(* Logix 5000 project; controller Transcat_L33ER vendor 1 type 14 code 107 rev 32.11; software revision 32.02; part 4 of 5 *)
(* tags used below, declared in another part *)
   AnyAutoDeviceInterlock : BOOL;   // Any device in Auto interlocked
   AnyAutoRun : BOOL;   // Bit that in on if ANY device is placed into Auto run (to signal pre-start beed)
   AnyDeviceInterlock : BOOL;   // Any device is interlocked
   AnyManualRun : BOOL;   // Bit that in on if ANY device is placed into manual run (to signal pre-start beed)
   Auto_Run_All_Interlock : BOOL;   // Bit to interlock all devices running in Auto
   BeaconBlueLight : ALIAS FOR TC_Remote_IO:3:O.3;   // Blue Beacon Light
   BeaconGreenLight : ALIAS FOR TC_Remote_IO:3:O.2;   // Green Beacon Light
   BeaconRedLight : ALIAS FOR TC_Remote_IO:3:O.0;   // Red Beacon Light
   BeaconYellowLight : ALIAS FOR TC_Remote_IO:3:O.1;   // Yellow Beacon Light
   Beep : BOOL;   // Bit to Activte Beacon Alarm
   BeepNew : ALIAS FOR TC_Remote_IO:3:O.4;
   Device : Device[20];
   EstopActive : BOOL;   // E
   EStopReset_OS : BOOL;   // Storage bit required by the ONS instruction
   EStopResetArmed : BOOL;   // Remembers that Banner entered the waiting-for-reset state
   EStopResetPulse : BOOL;   // One-scan pulse used to clear all 14 E-stop interlocks - allows reset of estop interlocks from physical reset button on V
   FT103 : BronkhorstFlowMeter;
   FT103B : BronkhorstFlowMeter;
   FT104 : BronkhorstFlowMeter;
   FT104B : BronkhorstFlowMeter;
   FT105 : BronkhorstFlowMeter;
   FT105B : BronkhorstFlowMeter;
   GF101 : Thayer_WB_Feeder;   // Thayer 1 Tags
   GF101_Write_Acknowledge : ALIAS FOR Thayer1_BS:O.Data[2].5;   // Thayer 1 (GF101) Acknowledge
   GF201 : Thayer_WB_Feeder;   // Thayer 2 Tags
   GF201_Write_Acknowledge : ALIAS FOR Thayer2_BS:O.Data[2].5;   // Thayer 2 (GF201) Acknowledge
   GreenFlashingOff : TIMER;
   GreenFlashingOn : TIMER;
   HMI_AllReset : BOOL;   // Bit to reset Auto/Man, AutoRun, RecipeRun, TimedRunEnable to 0 from HMI
   HMI_ProcessReset : BOOL;   // Bit to clear the process hold/inteerlock when all other device interlocks are cleared
   MX101 : Howes_Mixer;
   MX201 : Howes_Mixer;
   PT103_PV_RAW : ALIAS FOR TC_Remote_IO:1:I.Ch0Data;   // Raw (unscaled) pressure reading from PT103 - PSI * 100 (range 0 - 108 PSI)
   PT104_PV_RAW : ALIAS FOR TC_Remote_IO:1:I.Ch1Data;   // Raw (unscaled) pressure reading from PT104 - PSI * 100 (range 0 - 108 PSI)
   PT105_PV_RAW : ALIAS FOR TC_Remote_IO:1:I.Ch2Data;   // Raw (unscaled) pressure reading from PT105 - PSI * 100 (range 0 - 108 PSI)
   StartBeepTimer : TIMER;   // Timer to sound the beep alarm before starting a device
   VF101 : Acrison_Feeder;   // Medium Feeder Tags
   VF201 : Acrison_Feeder;   // Small Feeder 2 Tags
   VFD_Panel_Safety_Panel_Etop_OK : ALIAS FOR XS26_VFD_Cabinet_Safety_Controller:I1.Data[1].6;
   VFD_Panel_Safety_Remote_Estops_OK : ALIAS FOR XS26_VFD_Cabinet_Safety_Controller:I1.Data[1].7;
   VFD_Panel_Safety_WaitingForReset : ALIAS FOR XS26_VFD_Cabinet_Safety_Controller:I1.Data[1].5;
   YellowFlashOff : TIMER;
   YellowFlashOn : TIMER;
(* MainProgram, continued *)

ROUTINE InterlockLogic   (* ladder *)
// All interlock logic is handled here
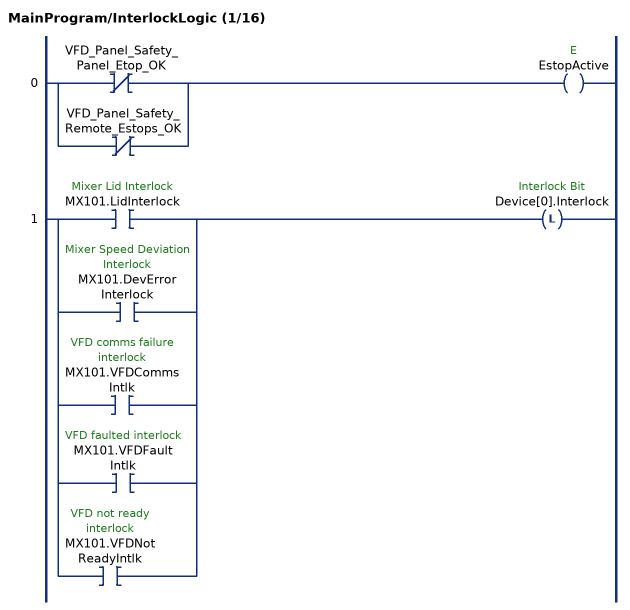
   0: [XIO(VFD_Panel_Safety_Panel_Etop_OK) ,XIO(VFD_Panel_Safety_Remote_Estops_OK) ]OTE(EstopActive);
   1: [XIC(MX101.LidInterlock) ,XIC(MX101.DevErrorInterlock) ,XIC(MX101.VFDCommsIntlk) ,XIC(MX101.VFDFaultIntlk) ,XIC(MX101.VFDNotReadyIntlk) ]OTL(Device[0].Interlock);
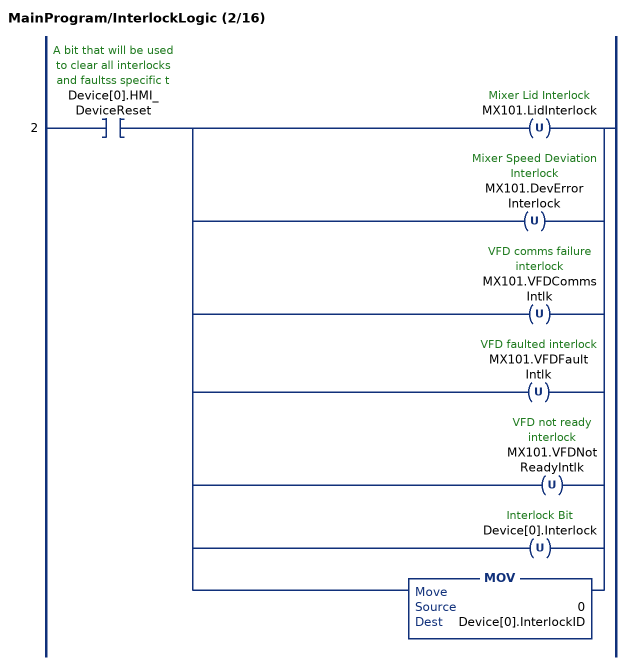
   2: XIC(Device[0].HMI_DeviceReset)[OTU(MX101.LidInterlock) ,OTU(MX101.DevErrorInterlock) ,OTU(MX101.VFDCommsIntlk) ,OTU(MX101.VFDFaultIntlk) ,OTU(MX101.VFDNotReadyIntlk) ,OTU(Device[0].Interlock) ,MOV(0,Device[0].InterlockID) ];
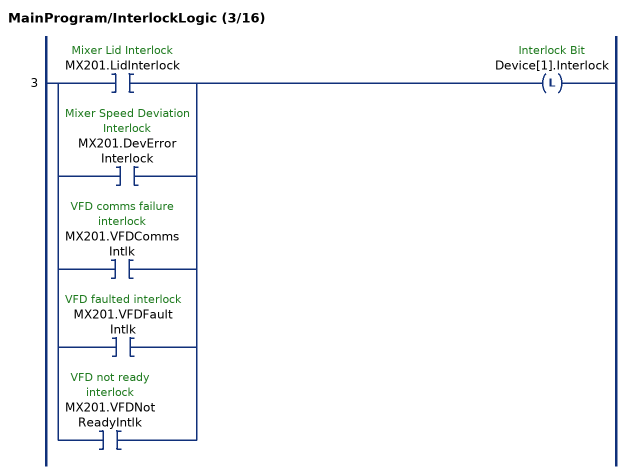
   3: [XIC(MX201.LidInterlock) ,XIC(MX201.DevErrorInterlock) ,XIC(MX201.VFDCommsIntlk) ,XIC(MX201.VFDFaultIntlk) ,XIC(MX201.VFDNotReadyIntlk) ]OTL(Device[1].Interlock);
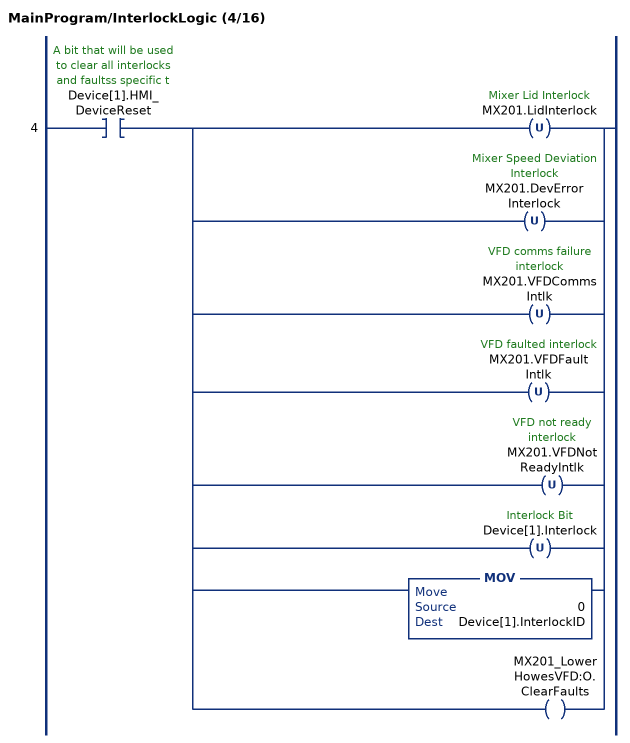
   4: XIC(Device[1].HMI_DeviceReset)[OTU(MX201.LidInterlock) ,OTU(MX201.DevErrorInterlock) ,OTU(MX201.VFDCommsIntlk) ,OTU(MX201.VFDFaultIntlk) ,OTU(MX201.VFDNotReadyIntlk) ,OTU(Device[1].Interlock) ,MOV(0,Device[1].InterlockID) ,OTE(MX201_LowerHowesVFD:O.ClearFaults) ];
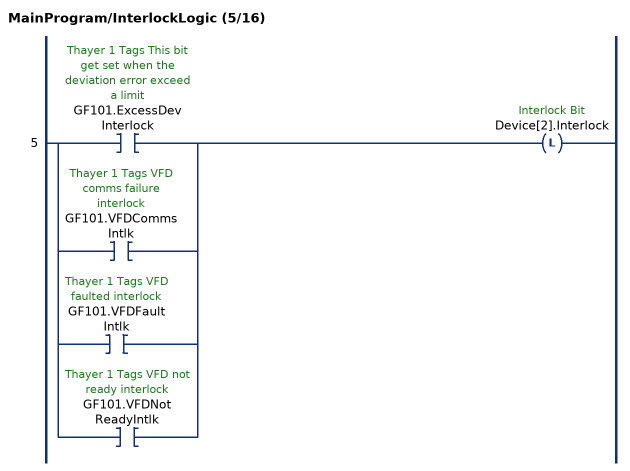
   5: [XIC(GF101.ExcessDevInterlock) ,XIC(GF101.VFDCommsIntlk) ,XIC(GF101.VFDFaultIntlk) ,XIC(GF101.VFDNotReadyIntlk) ]OTL(Device[2].Interlock);
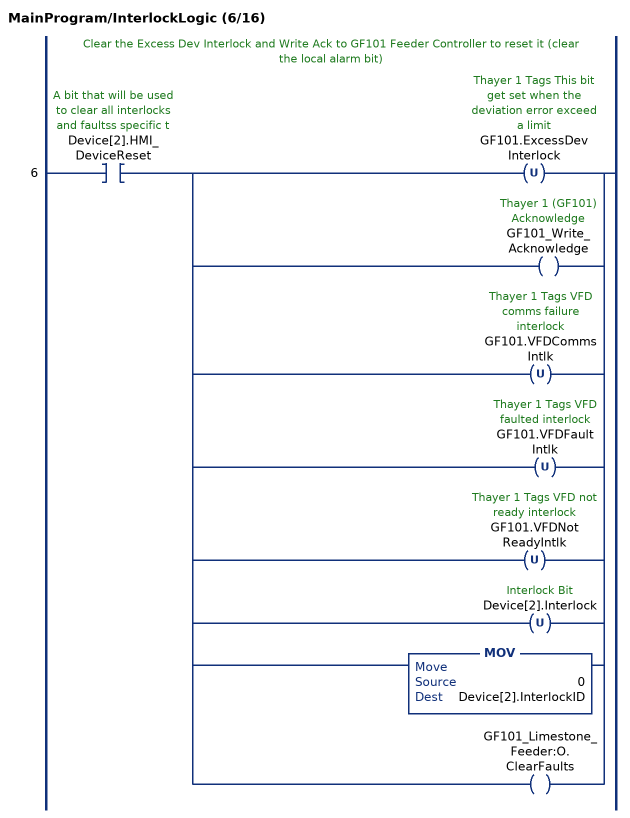
   // Clear the Excess Dev Interlock and Write Ack to GF101 Feeder Controller to reset it (clear the local alarm bit)
   6: XIC(Device[2].HMI_DeviceReset)[OTU(GF101.ExcessDevInterlock) ,OTE(GF101_Write_Acknowledge) ,OTU(GF101.VFDCommsIntlk) ,OTU(GF101.VFDFaultIntlk) ,OTU(GF101.VFDNotReadyIntlk) ,OTU(Device[2].Interlock) ,MOV(0,Device[2].InterlockID) ,OTE(GF101_Limestone_Feeder:O.ClearFaults) ];
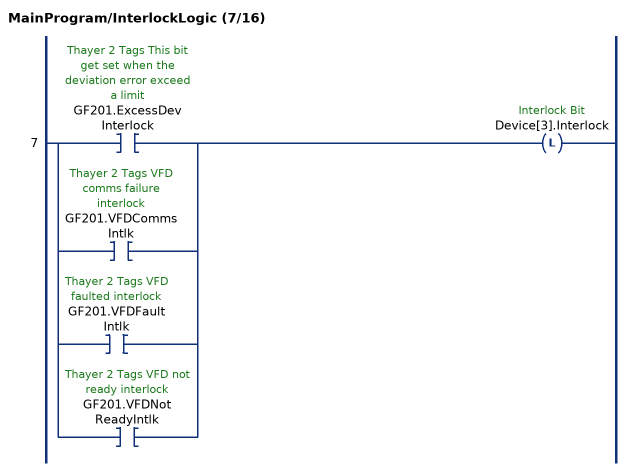
   7: [XIC(GF201.ExcessDevInterlock) ,XIC(GF201.VFDCommsIntlk) ,XIC(GF201.VFDFaultIntlk) ,XIC(GF201.VFDNotReadyIntlk) ]OTL(Device[3].Interlock);
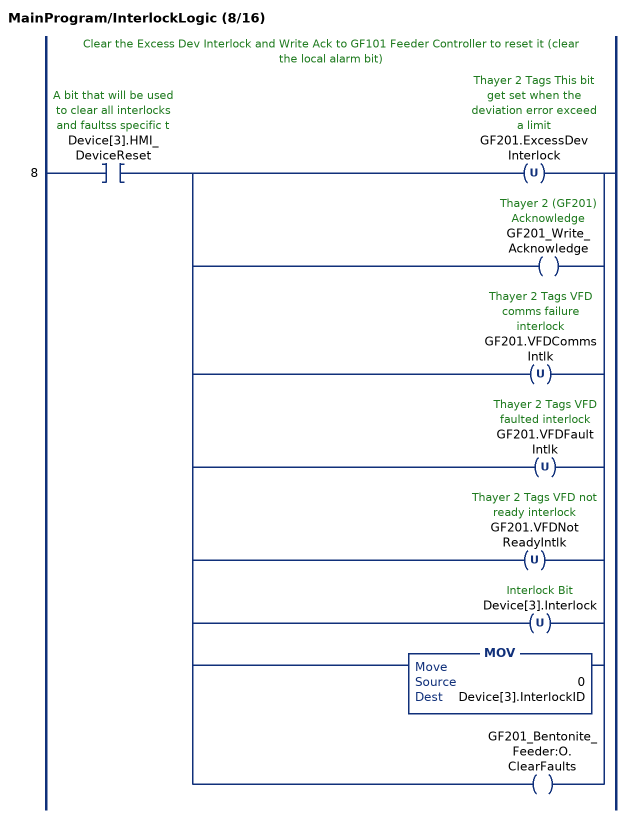
   // Clear the Excess Dev Interlock and Write Ack to GF101 Feeder Controller to reset it (clear the local alarm bit)
   8: XIC(Device[3].HMI_DeviceReset)[OTU(GF201.ExcessDevInterlock) ,OTE(GF201_Write_Acknowledge) ,OTU(GF201.VFDCommsIntlk) ,OTU(GF201.VFDFaultIntlk) ,OTU(GF201.VFDNotReadyIntlk) ,OTU(Device[3].Interlock) ,MOV(0,Device[3].InterlockID) ,OTE(GF201_Bentonite_Feeder:O.ClearFaults) ];
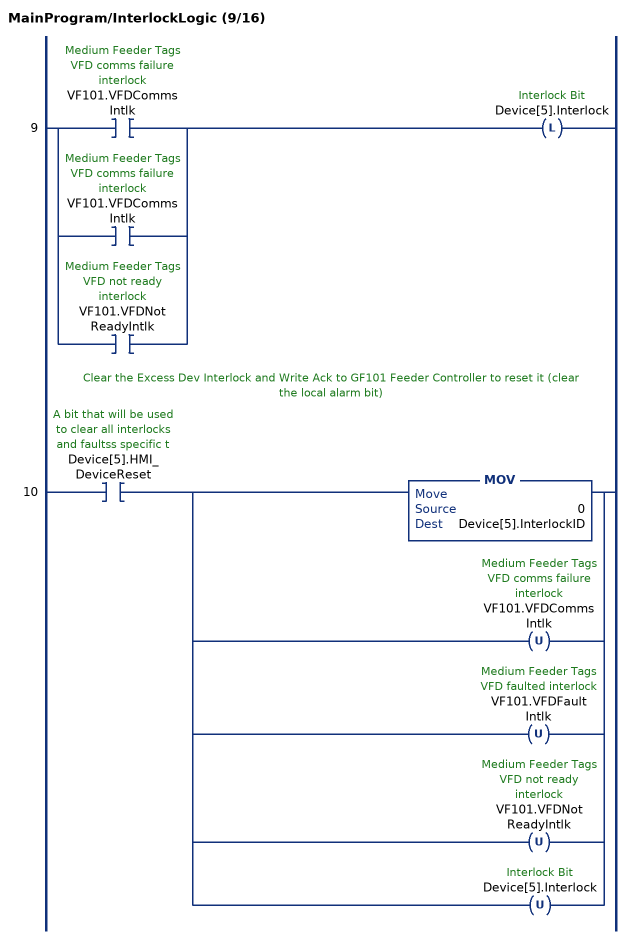
   9: [XIC(VF101.VFDCommsIntlk) ,XIC(VF101.VFDCommsIntlk) ,XIC(VF101.VFDNotReadyIntlk) ]OTL(Device[5].Interlock);
   // Clear the Excess Dev Interlock and Write Ack to GF101 Feeder Controller to reset it (clear the local alarm bit)
   10: XIC(Device[5].HMI_DeviceReset)[MOV(0,Device[5].InterlockID) ,OTU(VF101.VFDCommsIntlk) ,OTU(VF101.VFDFaultIntlk) ,OTU(VF101.VFDNotReadyIntlk) ,OTU(Device[5].Interlock) ];
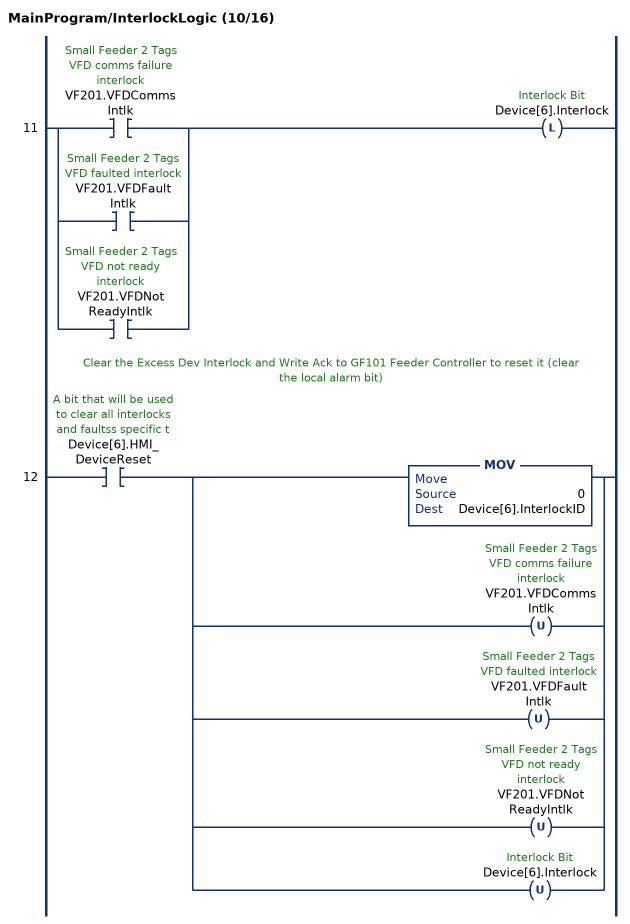
   11: [XIC(VF201.VFDCommsIntlk) ,XIC(VF201.VFDFaultIntlk) ,XIC(VF201.VFDNotReadyIntlk) ]OTL(Device[6].Interlock);
   // Clear the Excess Dev Interlock and Write Ack to GF101 Feeder Controller to reset it (clear the local alarm bit)
   12: XIC(Device[6].HMI_DeviceReset)[MOV(0,Device[6].InterlockID) ,OTU(VF201.VFDCommsIntlk) ,OTU(VF201.VFDFaultIntlk) ,OTU(VF201.VFDNotReadyIntlk) ,OTU(Device[6].Interlock) ];
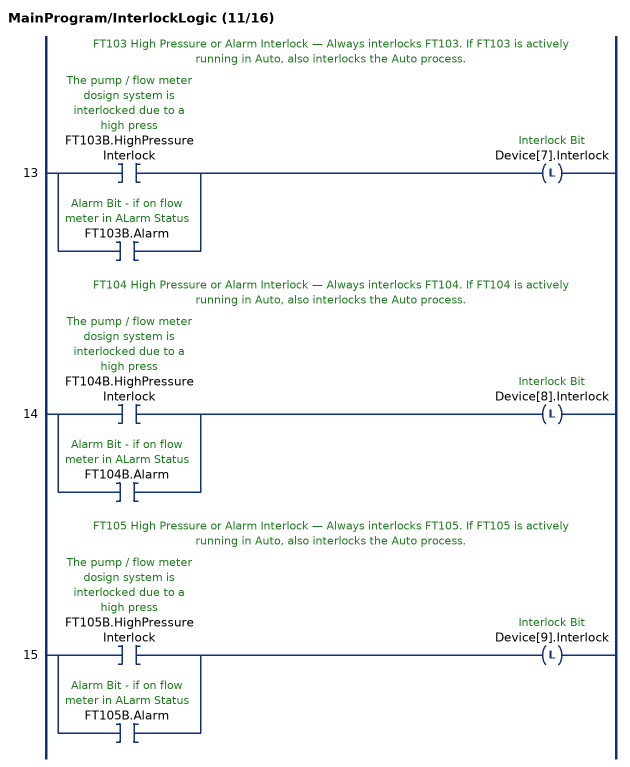
   // FT103 High Pressure or Alarm Interlock — Always interlocks FT103. If FT103 is actively running in Auto, also interlocks the Auto process.
   13: [XIC(FT103B.HighPressureInterlock) ,XIC(FT103B.Alarm) ]OTL(Device[7].Interlock);
   // FT104 High Pressure or Alarm Interlock — Always interlocks FT104. If FT104 is actively running in Auto, also interlocks the Auto process.
   14: [XIC(FT104B.HighPressureInterlock) ,XIC(FT104B.Alarm) ]OTL(Device[8].Interlock);
   // FT105 High Pressure or Alarm Interlock — Always interlocks FT105. If FT105 is actively running in Auto, also interlocks the Auto process.
   15: [XIC(FT105B.HighPressureInterlock) ,XIC(FT105B.Alarm) ]OTL(Device[9].Interlock);
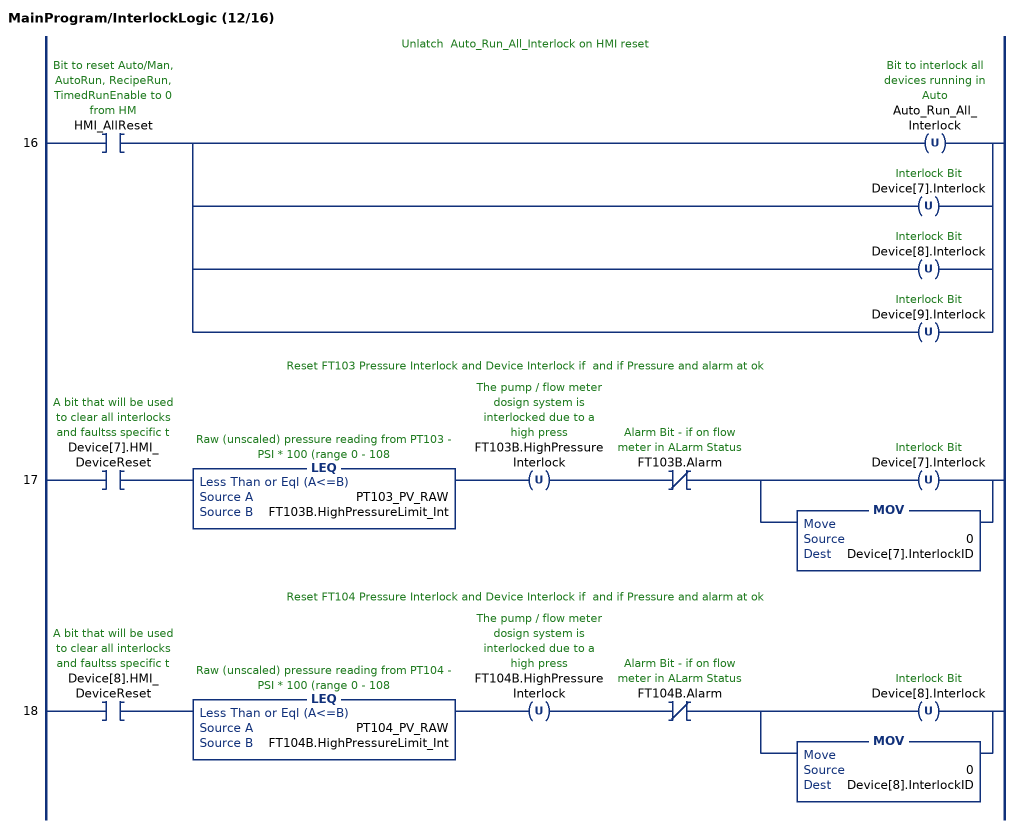
   // Unlatch  Auto_Run_All_Interlock on HMI reset
   16: XIC(HMI_AllReset)[OTU(Auto_Run_All_Interlock) ,[OTU(Device[7].Interlock) ,[OTU(Device[8].Interlock) ,OTU(Device[9].Interlock) ] ] ];
   // Reset FT103 Pressure Interlock and Device Interlock if  and if Pressure and alarm at ok
   17: XIC(Device[7].HMI_DeviceReset)LEQ(PT103_PV_RAW,FT103B.HighPressureLimit_Int)OTU(FT103B.HighPressureInterlock)XIO(FT103B.Alarm)[OTU(Device[7].Interlock) ,MOV(0,Device[7].InterlockID) ];
   // Reset FT104 Pressure Interlock and Device Interlock if  and if Pressure and alarm at ok
   18: XIC(Device[8].HMI_DeviceReset)LEQ(PT104_PV_RAW,FT104B.HighPressureLimit_Int)OTU(FT104B.HighPressureInterlock)XIO(FT104B.Alarm)[OTU(Device[8].Interlock) ,MOV(0,Device[8].InterlockID) ];
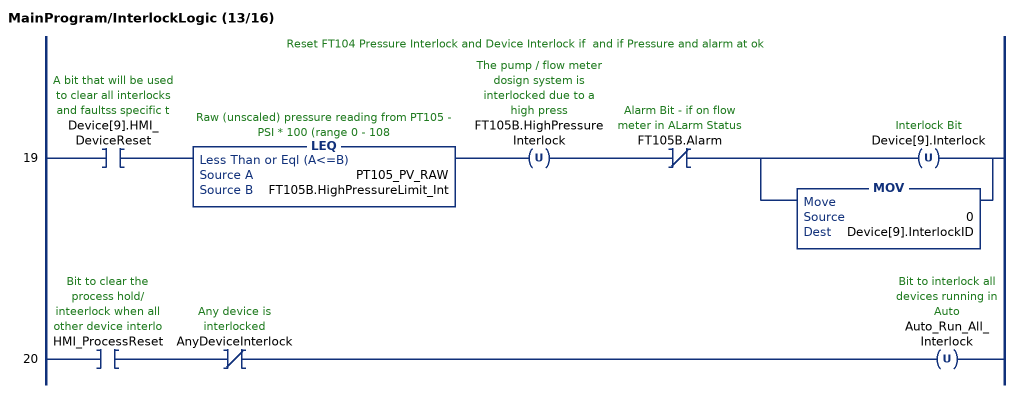
   // Reset FT104 Pressure Interlock and Device Interlock if  and if Pressure and alarm at ok
   19: XIC(Device[9].HMI_DeviceReset)LEQ(PT105_PV_RAW,FT105B.HighPressureLimit_Int)OTU(FT105B.HighPressureInterlock)XIO(FT105B.Alarm)[OTU(Device[9].Interlock) ,MOV(0,Device[9].InterlockID) ];
   20: XIC(HMI_ProcessReset)XIO(AnyDeviceInterlock)OTU(Auto_Run_All_Interlock);
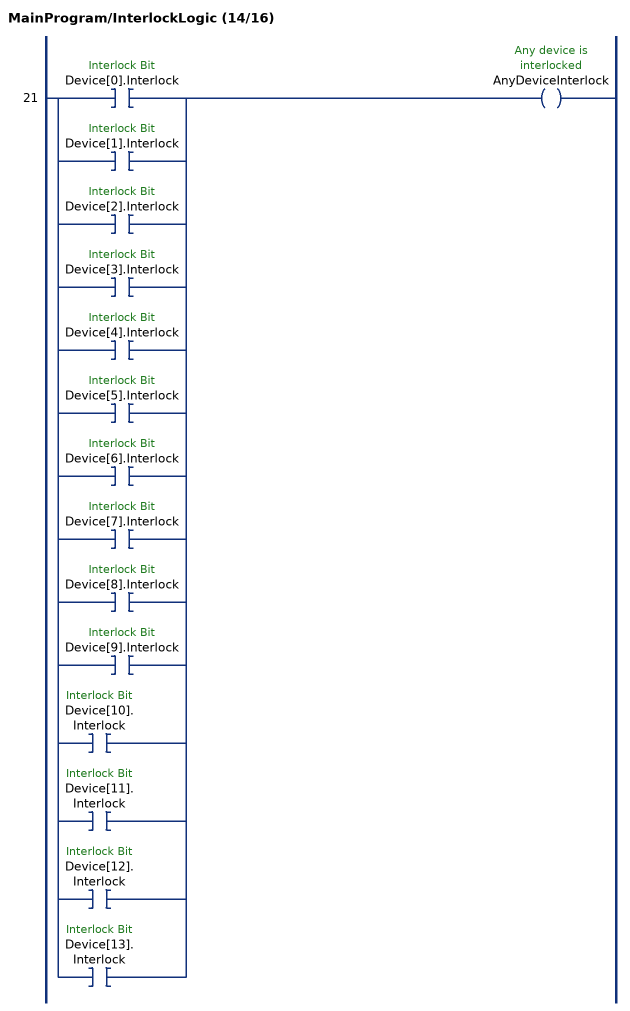
   21: [XIC(Device[0].Interlock) ,XIC(Device[1].Interlock) ,XIC(Device[2].Interlock) ,XIC(Device[3].Interlock) ,XIC(Device[4].Interlock) ,XIC(Device[5].Interlock) ,XIC(Device[6].Interlock) ,XIC(Device[7].Interlock) ,XIC(Device[8].Interlock) ,XIC(Device[9].Interlock) ,XIC(Device[10].Interlock) ,XIC(Device[11].Interlock) ,XIC(Device[12].Interlock) ,XIC(Device[13].Interlock) ]OTE(AnyDeviceInterlock);
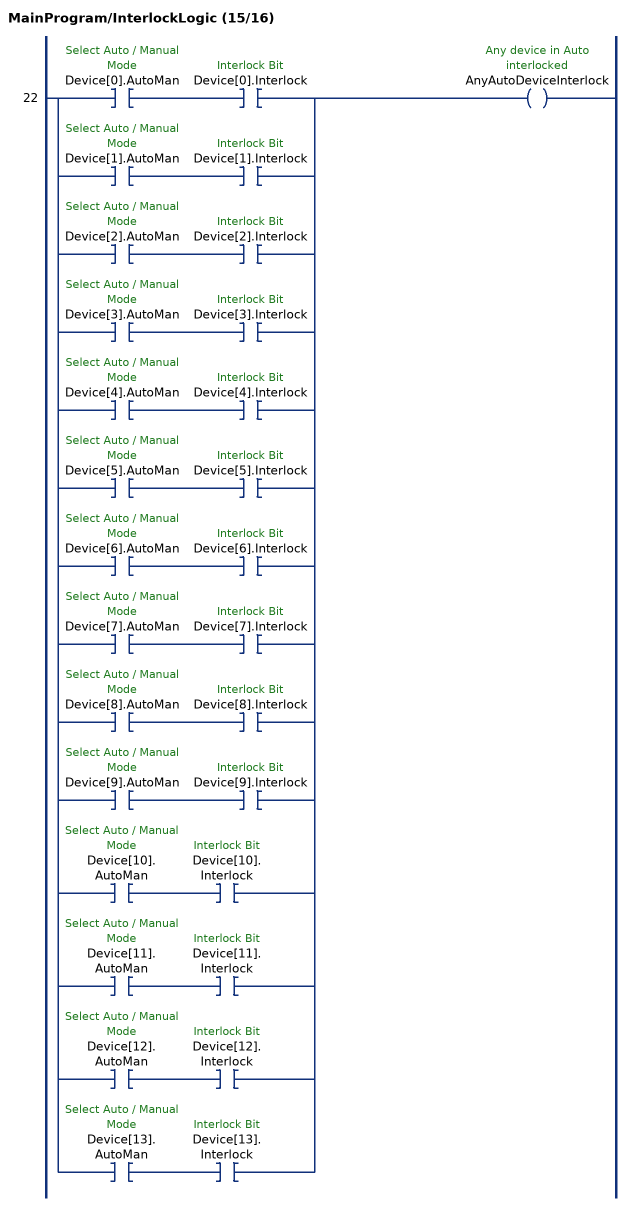
   22: [XIC(Device[0].AutoMan) XIC(Device[0].Interlock) ,XIC(Device[1].AutoMan) XIC(Device[1].Interlock) ,XIC(Device[2].AutoMan) XIC(Device[2].Interlock) ,XIC(Device[3].AutoMan) XIC(Device[3].Interlock) ,XIC(Device[4].AutoMan) XIC(Device[4].Interlock) ,XIC(Device[5].AutoMan) XIC(Device[5].Interlock) ,XIC(Device[6].AutoMan) XIC(Device[6].Interlock) ,XIC(Device[7].AutoMan) XIC(Device[7].Interlock) ,XIC(Device[8].AutoMan) XIC(Device[8].Interlock) ,XIC(Device[9].AutoMan) XIC(Device[9].Interlock) ,XIC(Device[10].AutoMan) XIC(Device[10].Interlock) ,XIC(Device[11].AutoMan) XIC(Device[11].Interlock) ,XIC(Device[12].AutoMan) XIC(Device[12].Interlock) ,XIC(Device[13].AutoMan) XIC(Device[13].Interlock) ]OTE(AnyAutoDeviceInterlock);
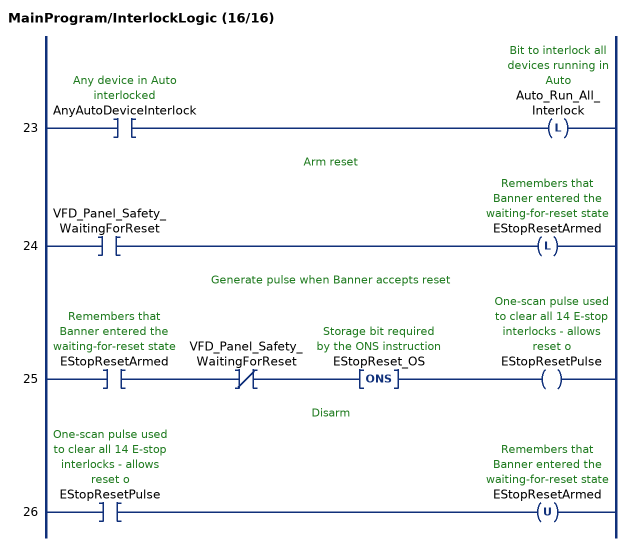
   23: XIC(AnyAutoDeviceInterlock)OTL(Auto_Run_All_Interlock);
   // Arm reset
   24: XIC(VFD_Panel_Safety_WaitingForReset)OTL(EStopResetArmed);
   // Generate pulse when Banner accepts reset
   25: XIC(EStopResetArmed)XIO(VFD_Panel_Safety_WaitingForReset)ONS(EStopReset_OS)OTE(EStopResetPulse);
   // Disarm
   26: XIC(EStopResetPulse)OTU(EStopResetArmed);
END_ROUTINE

ROUTINE Light_Beacon   (* ladder *)
// Indicator Light Beacon
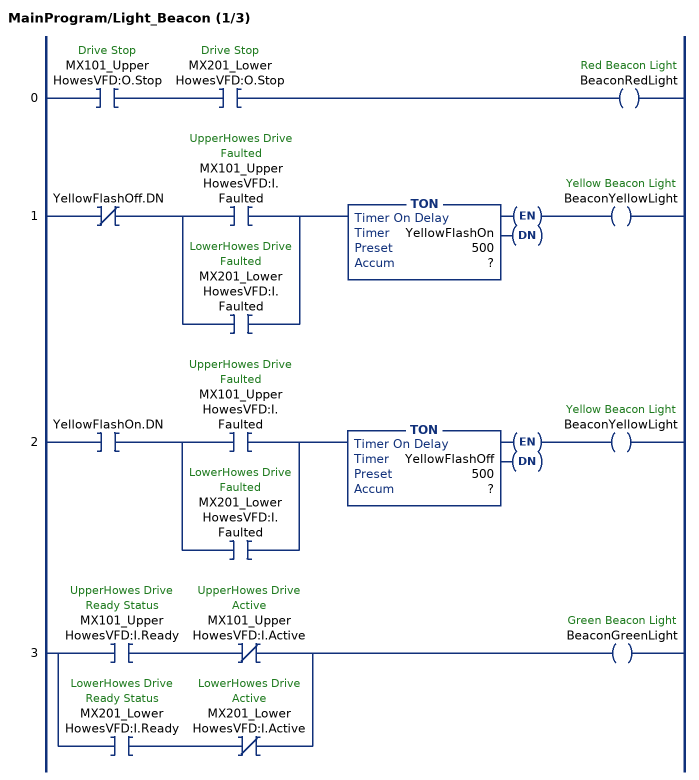
   0: XIC(MX101_UpperHowesVFD:O.Stop)XIC(MX201_LowerHowesVFD:O.Stop)OTE(BeaconRedLight);
   1: XIO(YellowFlashOff.DN)[XIC(MX101_UpperHowesVFD:I.Faulted) ,XIC(MX201_LowerHowesVFD:I.Faulted) ]TON(YellowFlashOn,?,?)OTE(BeaconYellowLight);
   2: XIC(YellowFlashOn.DN)[XIC(MX101_UpperHowesVFD:I.Faulted) ,XIC(MX201_LowerHowesVFD:I.Faulted) ]TON(YellowFlashOff,?,?)OTE(BeaconYellowLight);
   3: [XIC(MX101_UpperHowesVFD:I.Ready) XIO(MX101_UpperHowesVFD:I.Active) ,XIC(MX201_LowerHowesVFD:I.Ready) XIO(MX201_LowerHowesVFD:I.Active) ]OTE(BeaconGreenLight);
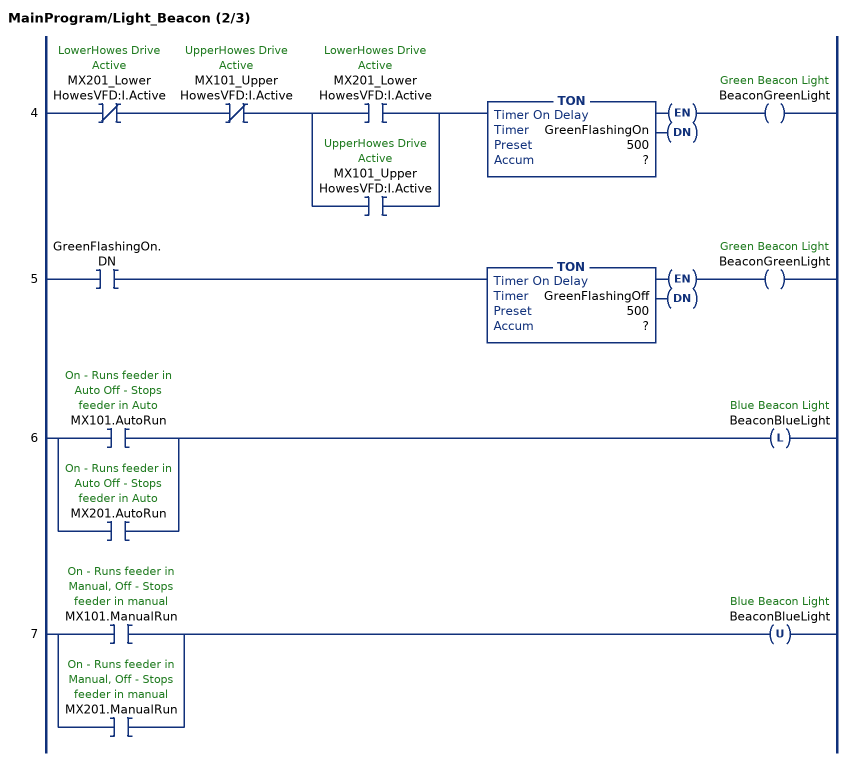
   4: XIO(MX201_LowerHowesVFD:I.Active)XIO(MX101_UpperHowesVFD:I.Active)[XIC(MX201_LowerHowesVFD:I.Active) ,XIC(MX101_UpperHowesVFD:I.Active) ]TON(GreenFlashingOn,?,?)OTE(BeaconGreenLight);
   5: XIC(GreenFlashingOn.DN)TON(GreenFlashingOff,?,?)OTE(BeaconGreenLight);
   6: [XIC(MX101.AutoRun) ,XIC(MX201.AutoRun) ]OTL(BeaconBlueLight);
   7: [XIC(MX101.ManualRun) ,XIC(MX201.ManualRun) ]OTU(BeaconBlueLight);
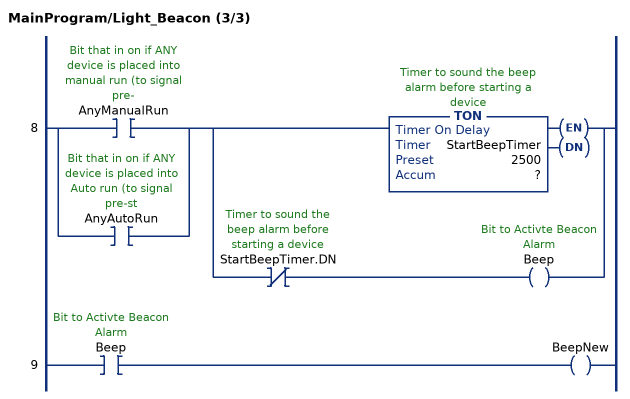
   8: [XIC(AnyManualRun) ,XIC(AnyAutoRun) ][TON(StartBeepTimer,?,?) ,XIO(StartBeepTimer.DN) OTE(Beep) ];
   9: XIC(Beep)OTE(BeepNew);
END_ROUTINE
